(* IEC 61131-3 sources: eCockpitGit/test_project/src/%F%00 Library/%F%JSON/%POU%FB_JSONWriter/%F%Structure, 4 files *)

(* ---- %METH%addKey.st ---- *)
//This adds a key and a value to the buffer
// |**Version**|**Author**| **Date** |**Changes**
// | 1         | NSN      | 22-06-20 | Creation
METHOD addKey : BOOL
VAR_INPUT
	name			:POINTER TO EASCII;	//Address of string for the tag name text
END_VAR
(*%!%__DELIMITER__%!%*)
IF ready AND NOT(afterKey OR inArray) AND inObject THEN
	addChar(char:=EASCII.DoubleQoute);
	addString(pString:=name);
	addChar(char:=EASCII.DoubleQoute);
	//Open tag ends
	addChar(char:=EASCII.Colon);
	afterKey			:=		TRUE;
	addKey				:=		TRUE;
END_IF

(* ---- %METH%arrayStart.st ---- *)
//This starts a new array
// |**Version**|**Author**| **Date** |**Changes**
// | 1         | NSN      | 22-06-20 | Creation
METHOD arrayStart : BOOL
VAR_INPUT
	singleLine		:BOOL;
END_VAR
(*%!%__DELIMITER__%!%*)
IF ready AND (afterKey OR inArray) AND treeLevel < levelsMax THEN
	//Struct tag starts
	addChar(char:=EASCII.SqBracketO);
	treeLevel					:=		treeLevel + 1;
	treeTypes[treeLevel]		:=		EStructType.tArray;
	treeSingleLine[treeLevel]	:=		singleLine;
	//New Line
	IF NOT(useSingleLine) AND NOT(treeSingleLine[treeLevel]) THEN
		addNewLine();
	END_IF
	inArray						:=		TRUE;
	afterKey					:=		FALSE;
	inObject					:=		FALSE;
	arrayStart					:=		TRUE;
	emptyBlock					:=		TRUE;
END_IF

(* ---- %METH%objectStart.st ---- *)
//This starts a new object
// |**Version**|**Author**| **Date** |**Changes**
// | 1         | NSN      | 22-06-20 | Creation
METHOD objectStart : BOOL
VAR_INPUT
	singleLine		:BOOL;
END_VAR
(*%!%__DELIMITER__%!%*)
IF ready AND (afterKey OR inArray) AND treeLevel < levelsMax THEN
	//Struct tag starts
	addChar(char:=EASCII.OpenBraces);
	treeLevel					:=		treeLevel + 1;
	treeTypes[treeLevel]		:=		EStructType.object;
	treeSingleLine[treeLevel]	:=		singleLine;
	//New Line
	IF NOT(useSingleLine) AND NOT(treeSingleLine[treeLevel]) THEN
		addNewLine();
	END_IF
	afterKey					:=		FALSE;
	inArray						:=		FALSE;
	inObject					:=		TRUE;
	objectStart					:=		TRUE;
	emptyBlock					:=		TRUE;
END_IF

(* ---- %METH%structEnd.st ---- *)
//This ends the previously started object
// |**Version**|**Author**| **Date** |**Changes**
// | 1         | NSN      | 22-06-20 | Creation
METHOD structEnd : BOOL
VAR
	moveCommaBuffer		:POINTER TO EASCII;
END_VAR
(*%!%__DELIMITER__%!%*)
IF ready AND treeLevel > 0 AND treeTypes[treeLevel] = EStructType.object OR treeTypes[treeLevel] = EStructType.tArray THEN
	IF afterKey THEN
		writeNull();
	END_IF
	IF NOT(emptyBlock) THEN
		IF lastComma <> 0 THEN
			WHILE lastComma < bufferPosition DO
				moveCommaBuffer		:=		lastComma + 1;
				lastComma^			:=		moveCommaBuffer^;
				lastComma			:=		lastComma + 1;
			END_WHILE
			bufferPosition			:=		bufferPosition - 1;
			lastComma				:=		0;
		END_IF
	END_IF
	//Last TAB is deleted
	IF NOT(useSingleLine) AND NOT(treeSingleLine[treeLevel]) THEN
		bufferPosition			:=		bufferPosition - 1;
	END_IF
	//struct tag ends
	CASE treeTypes[treeLevel] OF
		EStructType.tArray:
			addChar(char:=EASCII.SqBracketC);
		EStructType.object:
			addChar(char:=EASCII.CloseBraces);
	END_CASE
	lastComma					:=		bufferPosition;
	addChar(char:=EASCII.Comma);
	treeLevel					:=		treeLevel - 1;
	IF treeLevel > 0 THEN
		IF NOT(useSingleLine) AND NOT(treeSingleLine[treeLevel]) THEN
			addNewLine();
		END_IF
		CASE treeTypes[treeLevel] OF
			EStructType.tArray:
				inArray			:=		TRUE;
				inObject		:=		FALSE;
			EStructType.object:
				inObject		:=		TRUE;
				inArray			:=		FALSE;
		END_CASE
	END_IF
	structEnd					:=		TRUE;
	emptyBlock					:=		FALSE;
END_IF
